# EPICS autosave request: iocBoot/sioc-esb-xps4/xps.req
file xpsm.req P=ESB:XPS4:m1
file xpsm.req P=ESB:XPS4:m2
file xpsm.req P=ESB:XPS4:m3
file xpsm.req P=ESB:XPS4:m4
file xpsm.req P=ESB:XPS4:m5
file xpsm.req P=ESB:XPS4:m6
file xpsm.req P=ESB:XPS4:m7
file xpsm.req P=ESB:XPS4:m8
ESB:XPS4:MOVE:INC
